// TIA Portal V20 export
TYPE "UDT_PartPosition"
   STRUCT
      Undrilled : Struct
         Presence : "UDT_PartPresence";
         States : "UDT_PartStates";
      END_STRUCT;
      Drilled : Struct
         Presence : "UDT_PartPresence";
         States : "UDT_PartStates";
      END_STRUCT;
   END_STRUCT;
END_TYPE
